(*
    Single integration smoke for FB_REF. Goal: prove the FB_REF wiring
    (REFERENCE TO refs, CallAfterInit / CallAfterInitEx / CallAfterInitExEx
    chain, inline-init of fbStates, per-state name/fDelta defaults,
    PMPS state-key registration) still drives FB_MotionStageNC into the
    configured fPosition for a commanded state.

    The motion-stack itself (FB_MotionStageNC, FB_PositionStatePMPSND,
    FB_StateSetup, FB_AtPositionState, ...) is fully covered by the
    lcls-twincat-motion-abstraction test suite. This test only checks
    that the CC FB_REF wrapper does not break the contract.

    Procedure:
        1. Wait for first-scan motor setup + PMPS DB loaded.
        2. Command IN (configured fPosition = 20.0, fDelta = 2.0).
        3. Wait for eEnumGet = IN AND |fActPosition - 20.0| <= fDelta.
        4. TEST_FINISHED.
    On watchdog expiry: AssertTrue(FALSE, ...) with the step + observed
    eEnumGet + observed fActPosition so the failure mode is obvious in
    the TcUnit log.
*)
{attribute 'analysis' := '-33'}
FUNCTION_BLOCK FB_REFTest EXTENDS FB_TestSuite
VAR
    axRef    : AXIS_REF;
    fbPDS    : LCLS_Tc_DevAbs.FB_PersistentDataStorage;

    fbMotorY : FB_MotionStageNC(AxisRef := axRef, iPersistentDataStorage := fbPDS, sName := 'Y');


    aiMotionStage : ARRAY[1..MotionConstants.MAX_STATE_MOTORS] OF I_MotionStage := [fbMotorY];

    {attribute 'pytmc' := '
        pv: MMS
        astPositionState.array: 1..2
    '}
    astPositionState : ARRAY[1..MotionConstants.MAX_STATE_MOTORS]
                         OF ARRAY[1..GeneralConstants.MAX_STATES] OF ST_PositionState;

    fbFFHWO    : FB_HardwareFFOutput;
    fbArbiter  : FB_Arbiter(1);
    fbSubSysIO : FB_DummyArbIO;

    bEnableMotion         : BOOL;
    bEnableBeamParams     : BOOL;
    bEnablePositionLimits : BOOL;
    bReadDBNow            : BOOL;

    sDeviceName    : STRING := 'TST:REF';
    sTransitionKey : STRING := 'TST:REF-TRANSITION';

    stDefault : ST_PositionState := (
        bMoveOk       := TRUE,
        bValid        := TRUE,
        bUseRawCounts := FALSE
    );

    afbStatePMPS : ARRAY[1..2] OF FB_CC_StatePMPSConfig[
        (stPositionState := astPositionState[1][E_REF_States.OUT],
         stDefault       := stDefault,
         fPosition       := 10.0,
         sPmpsState      := 'TST:REF-OUT'),
        (stPositionState := astPositionState[1][E_REF_States.IN],
         stDefault       := stDefault,
         fPosition       := 20.0,
         sPmpsState      := 'TST:REF-IN')
    ];

    fbREF : FB_REF(
        aiMotionStage    := aiMotionStage,
        astPositionState := astPositionState,
        fbFFHWO          := fbFFHWO,
        fbArbiter        := fbArbiter,
        sDeviceName      := sDeviceName,
        sTransitionKey   := sTransitionKey
    ) := ( MaintMode := TRUE) ;

    fbTestTimer : TON := (IN := TRUE, PT := T#120S);
    nTestStep   : INT;
    fGoal       : LREAL := 20.0;
    fTolerance  : LREAL := 2.0;
    fObserved   : LREAL;
    bFirstScan : BOOL := TRUE;
    i	: UINT;
END_VAR

TEST(__POUNAME());

CASE nTestStep OF
    0:

        IF bFirstScan THEN
            fbMotorY.SetModeEnableLimits(
                LimBackward    := TRUE,
                LimForward     := TRUE,
                HomeEnable     := FALSE,
                BrakeMode      := E_StageBrakeMode.IF_ENABLED,
                EnableMode     := E_StageEnableMode.DURING_MOTION,
                HomeMode       := E_EpicsHomeCmd.LOW_LIMIT,
                UserEnable     := TRUE,
                HardwareEnable := TRUE
            );
            fbMotorY.SetVelocity(Velocity := 15.5);
            fbMotorY.RestoreMotionParams      := FALSE;
            fbMotorY.DoNotRestoreNcParameters := TRUE;

            bEnableMotion         := TRUE;
            bEnableBeamParams     := TRUE;
            bEnablePositionLimits := TRUE;
            bReadDBNow            := TRUE;
            fbREF(
                bFileReaderBusy  := TRUE,
                bFileReaderError := FALSE
            );
            bFirstScan := FALSE;

        END_IF
        nTestStep      := 1;
    1:
        fbREF(
            bFileReaderBusy  := FALSE,
            bFileReaderError := FALSE
        );
        nTestStep      := 2;
    2:
        (* Wait for cold-start stabilisation: PMPS DB parsed, motor
           ready to accept moves, no residual error. *)
        IF fbMotorY.stMotionStatus.bStageReady
           AND NOT fbMotorY.stMotionStatus.bError THEN
            fbREF.eEnumSet := E_REF_States.IN;
            nTestStep      := 3;
        END_IF

    3:
        fObserved := fbMotorY.stMotionStatus.fActPosition;
        IF fbREF.eEnumGet = E_REF_States.IN
           AND NOT fbMotorY.stMotionStatus.bMoving
           AND ABS(fObserved - fGoal) <= fTolerance THEN
            AssertTrue(
                Condition := TRUE,
                Message   := 'T01: REF reached IN within tolerance');
            nTestStep := 4;
        END_IF
END_CASE

// FOR i := 1 TO 2 DO
//     afbStatePMPS[i]();
// END_FOR

fbPDS();
fbMotorY();

fbREF(
    bEnableMotion         := bEnableMotion,
    bEnableBeamParams     := bEnableBeamParams,
    bEnablePositionLimits := bEnablePositionLimits,
    bReadDBNow            := bReadDBNow
);

fbSubSysIO(LA := fbArbiter, FFO := fbFFHWO);
fbTestTimer();

IF nTestStep = 10 THEN
    TEST_FINISHED();
ELSIF fbTestTimer.Q THEN
    AssertTrue(
        Condition := FALSE,
        Message   := CONCAT(
            CONCAT(
                CONCAT('T01: timed out at step ', TO_STRING(nTestStep)),
                CONCAT(', eEnumGet=', TO_STRING(TO_UDINT(fbREF.eEnumGet)))),
            CONCAT(', fActPos=', TO_STRING(fObserved))));
    TEST_FINISHED();
END_IF

(*
    Wiring smoke for FB_REF. Commands IN (configured fPosition = 20.0)
    and asserts (a) eEnumGet reports IN and (b) the Y motor's actual
    position lands within fDelta (2.0) of the configured set point.

    Watchdog: 60s. Fail message includes the step number, the observed
    eEnumGet, and the observed fActPosition so a failure points at
    which part of the wiring chain broke.
*)
METHOD PRIVATE T01_StateMove_RequestIn_MotorReachesConfiguredPosition
VAR_INST

END_VAR
END_METHOD

END_FUNCTION_BLOCK

(* stored: Version 1.1.0.1
   POU FB_REFTest: Id {bc00a2b4-c887-49cb-85f5-b51e5f3fe97d}, SpecialFunc None
   Method T01_StateMove_RequestIn_MotorReachesConfiguredPosition: Id {bc00a201-0000-0000-0000-000000000001} *)
